// TIA Portal V18 export
// export: Created 2026-06-22T15:41:34.8993659Z, ExportSetting WithDefaults, DisplayName Totally Integrated Automation Portal, DisplayVersion V18, DisplayName TIA Portal Openness, DisplayVersion V18, DisplayName TIA Portal Version Control Interface, DisplayVersion V18, DisplayName STEP 7 Professional, DisplayVersion V18, DisplayName STEP 7 Safety, DisplayVersion V18, DisplayName WinCC Professional, DisplayVersion V18
VAR_GLOBAL   // PLC tag table "PLC2_Tags"
   MB_ControlWord AT %MW40 : Word;
   MB_FreqSetpoint AT %MW42 : Int;
   MB_StatusWord AT %MW44 : Word;
   MB_ActualSpeed AT %MW46 : Int;
   MB_Error AT %M50.0 : Bool;
   MB_Busy AT %M50.1 : Bool;
   MB_Done AT %M50.2 : Bool;
   MB_Status AT %MW52 : Word;
   iStep AT %MW60 : Int;
   Freq_Temp AT %MD70 : Real;
   Speed_Actual_Temp AT %MD74 : Real;
   FirstScan AT %M101.0 : Bool;
   Clock_1Hz AT %M100.5 : Bool;
   MBCL_Done AT %M51.0 : Bool;
   MBCL_Error AT %M51.1 : Bool;
   MBCL_Status AT %MW54 : Word;
END_VAR
